FUNCTION_BLOCK ARRAY2VALUES_2_LREAL (* Service Interface Function Block Type *)
  PACKAGE eclipse4diac::convert;
  {SET_ATTRIBUTE(eclipse4diac::core::GenericClassName, 'GEN_ARRAY2ARRAY')}
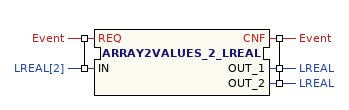
  EVENT_INPUT
    REQ WITH IN; (* Service Request *)
  END_EVENT
  EVENT_OUTPUT
    CNF WITH OUT_1, OUT_2; (* Confirmation of Requested Service *)
  END_EVENT
  VAR_INPUT
    IN : ARRAY [0..1] OF LREAL; (* Array input *)
  END_VAR
  VAR_OUTPUT
    OUT_1 : LREAL; (* output number 1 *)
    OUT_2 : LREAL; (* output number 2 *)
  END_VAR
END_FUNCTION_BLOCK
